Staubli VAL3: reset.pgx

public program reset()
  local num i
  local string l_sName
  local num l_nPos
  local string l_sKey
begin
  // scan it
  l_sKey=first(pt:tTraj)
  while l_sKey!=""
    if l_sKey!=""
      pt:tTraj[l_sKey].nIndex=0
    endIf
    l_sKey=next(pt:tTraj[l_sKey])
  endWhile
  // exit
end
